Universal Robots PolyScope program: path_straight_line.urp

Program path_straight_line (installation=default directory=/programs/andyl createdIn=5.11.9.1010452 lastSavedIn=5.11.9.1010452 robotSerialNumber=20225200364)
Calibrated DH parameters: a=[0.00002, -0.569483, -0.54992, -0.00001, -0.000036, 0]; d=[0.180894, -146.691669, 192.918669, -46.053088, 0.119778, 0.115602]; alpha=[1.571425, -0.001534, 0.003359, 1.568739, -1.571477, 0]; deltaTheta=[0, 0.376258, -0.101074, -0.275185, -0.000002, 0]
Robot Program (runOnlyOnce=true)
  Script file /programs/andyl/script_snippets/start_onrobot_ft_rtde_export_thread.script
    | # UR10e demo-1.2: non-blocking OnRobot Variables RTDE export.
    | # Insert this as a PolyScope Script node near the start of the program.
    | # It continuously writes the OnRobot URCap variables Fx/Fy/Fz/Tx/Ty/Tz
    | # into RTDE output_double_register_24..29 while the program runs.
    | 
    | thread onrobot_ft_rtde_export_thread():
    |   while True:
    |     write_output_float_register(24, Fx)
    |     write_output_float_register(25, Fy)
    |     write_output_float_register(26, Fz)
    |     write_output_float_register(27, Tx)
    |     write_output_float_register(28, Ty)
    |     write_output_float_register(29, Tz)
    |     sync()
    |   end
    | end
    | 
    | global onrobot_ft_rtde_export_handle = run onrobot_ft_rtde_export_thread()
  Script file /programs/andyl/script_snippets/approach_above_path_start.script
    | # UR10e demo-1.2: approach above the recorded F/T Path start.
    | # Use this from a PolyScope Script node before F/T Search.
    | # It keeps the current TCP Z, aligns X/Y/orientation to the path home pose,
    | # then moves slowly with movel. It does not execute any force search.
    | 
    | path_home_x = 0.4447489624
    | path_home_y = 0.2284111481
    | path_home_z = 0.0195379200
    | path_home_rx = 3.1415727139
    | path_home_ry = -0.0000264648
    | path_home_rz = -0.0000241579
    | 
    | start_pose = get_actual_tcp_pose()
    | safe_min_z = path_home_z + 0.010
    | 
    | if start_pose[2] < safe_min_z:
    |   popup("Start TCP is too low for XY approach. Move up first.", title="Approach guard", error=True, blocking=True)
    |   halt
    | end
    | 
    | approach_pose = p[path_home_x, path_home_y, start_pose[2], path_home_rx, path_home_ry, path_home_rz]
    | textmsg("approach_above_path_start target: ", approach_pose)
    | movel(approach_pose, a=0.05, v=0.04)
  URCap F/T Zero (FT-OnRobot, OnRobot A/S)
  URCap F/T Guard (FT-OnRobot, OnRobot A/S) dataModel(OF_PID=0, coordsys=1, advanced=false, absolute=true, FX=0.0, FY=0.0, FZ=0.0, TX=0.0, TY=0.0, TZ=0.0, F3D=50.0, T3D=1.0, INDEX=0, STATE=true)
    URCap F/T Search (FT-OnRobot, OnRobot A/S) dataModel(type=1, coordsys=1, speed=0.01, acceleration=0.5, rpy=[0.0, 0.0, 0.0], popupLimit=true, ftarray=[0.0, 0.0, 0.0, 0.0, 0.0, 0.0, 2.0, 0.0], ftabsarray=[false, false, false, false, false, false])
      URCap F/T Waypoint (FT-OnRobot, OnRobot A/S) dataModel(pose=p[0.4459648348526117,0.22972055741315447,0.03182057305993935,3.1414720887816623,-8.345103664906338E-5,-4.277820267408178E-5], type=2, z=0.05, variable=B2Empty)
    URCap F/T Control (FT-OnRobot, OnRobot A/S) dataModel(coordsys=1, enarray=[false, false, true, false, false, false], useAdvancedParameters=true, ftarray=[0.0, 0.0, 5.0, 0.0, 0.0, 0.0], gains=[0.5, 0.1, 0.1, 0.1, 0.0, 0.0])
      URCap F/T Move (FT-OnRobot, OnRobot A/S) dataModel(type=0, speed=0.01, acceleration=0.5, rpy=[0.0, 0.0, 0.0], popupLimit=true, ftarray=[0.0, 0.0, 0.0, 0.0, 0.0, 0.0, 0.0, 0.0], ftabsarray=[false, false, false, false, false, false])
        URCap F/T Path (FT-OnRobot, OnRobot A/S) dataModel(path_id=3964, type=1)
    Script file /programs/andyl/script_snippets/retract_after_ft_path_tool_minus_z.script
      | # UR10e demo-1.2: automatic retract after F/T Control + F/T Path.
      | # Assumption for the current program: F/T Search contacts along Tool +Z,
      | # so retracting along Tool -Z moves away from the surface.
      | 
      | retract_distance = -0.020
      | retract_speed = 0.010
      | retract_acc = 0.050
      | 
      | retract_start_pose = get_actual_tcp_pose()
      | retract_target_pose = pose_trans(retract_start_pose, p[0, 0, retract_distance, 0, 0, 0])
      | 
      | textmsg("retract_after_ft_path_tool_minus_z start: ", retract_start_pose)
      | textmsg("retract_after_ft_path_tool_minus_z target: ", retract_target_pose)
      | 
      | movel(retract_target_pose, a=retract_acc, v=retract_speed)
